INTERFACE ITF_ControlElement_HMI_Connector_1 EXTENDS ITF_BaseControlElement_HMI_Connector

END_INTERFACE

(* stored: Version 1.1.0.1, ProductVersion 3.1.4024.15
   Itf ITF_ControlElement_HMI_Connector_1: Id {36d8e96d-f495-45f9-a575-70f7a488fbfc} *)
